TYPE (* Typedef of the non-TP CAN Message (0..8 Byte only) *)
  (* Version 1.0, 2025-09-04, Franz Höpfinger, initial API and implementation and/or initial documentation *)
  PACKAGE isobus::pgn;
  IMPORT eclipse4diac::core::TypeHash;
  CAN_MSG : STRUCT
    u16DaSize : UINT := 0; (* Number of bytes recorded (0..8) *)
    u8Priority : USINT := 7; (* Priority (0..7) 0=highest *)
    data : ARRAY [0..7] OF BYTE := [16#FF, 16#FF, 16#FF, 16#FF, 16#FF, 16#FF, 16#FF, 16#FF]; (* data buffer *)
  END_STRUCT;
END_TYPE
